FUNCTION_BLOCK RunCableHolder EXTENDS RunUnitSlave
VAR
	//devices
	holderFixedEnd : POINTER TO RunCylinder;
	holderMovingEnd : POINTER TO RunCylinder;
	shifterShort : POINTER TO RunCylinder;
	shifterLong : POINTER TO RunCylinder;
	//axis (share
	axis : POINTER TO RunAxis;
	ptDrag : POINTER TO ParameterSet;
	ptRelease : pointer to ParameterSet;
END_VAR

SUPER^();

CASE outputState OF
	//---------------Initialize
	eSpecialStates.INITIAL_BEGIN:
		transitionByte.0 :=  holderFixedEnd^.Execute(eCylinderCommands.COMMAND_A);
		transitionByte.1 :=  holderMovingEnd^.Execute(eCylinderCommands.COMMAND_A);
		transitionByte.2 :=  shifterShort^.Execute(eCylinderCommands.COMMAND_A);
		transitionByte.3 :=  shifterLong^.Execute(eCylinderCommands.COMMAND_A);
		IF transitionByte = 16#F THEN
			NextState := eSpecialStates.INITIAL_END;
		END_IF
	//---------------Working
	eSpecialStates.SLAVE_ENTER_PROCEDURE:
		IF SlotBase^.Valid THEN
			bSerialTransition := TRUE;
		ELSE
			NextState := eSpecialStates.SLAVE_WORK_DONE;	
		END_IF
		//TODO , check ok/ng?
	16#201:
		bSerialTransition := shifterLong^.Execute(eCylinderCommands.COMMAND_B);
	16#202:
		//hold
		transitionByte.0 :=  holderFixedEnd^.Execute(eCylinderCommands.COMMAND_B);
		transitionByte.1 :=  holderMovingEnd^.Execute(eCylinderCommands.COMMAND_B);
		bSerialTransition := (transitionByte = 16#3);
	16#203:
		bSerialTransition := axis^.ExecuteParameter(ptDrag);//inform transporter moving work2
	16#204:
		//strech
		IF shifterShort^.Execute(eCylinderCommands.COMMAND_B) THEN
			slaveWorkingSignal[1] := TRUE; //inform to labeler handler to work
			NextState := 16#210;
		END_IF
	//-------------Releasing
	16#210:
		//wait until
		bSerialTransition := NOT slaveWorkingSignal[1];
	16#211:
		transitionByte.0 := holderFixedEnd^.Execute(eCylinderCommands.COMMAND_A); //release
		transitionByte.1 := holderMovingEnd^.Execute(eCylinderCommands.COMMAND_A);
		IF transitionByte = 16#3 THEN
			bSerialTransition := TRUE;
		END_IF
	16#212:
		bSerialTransition := axis^.ExecuteParameter(ptRelease);//inform transporter moving release
	16#213:
		//release
		bSerialTransition := shifterLong^.Execute(eCylinderCommands.COMMAND_A);
	16#214:
		//release
		bSerialTransition := holderMovingEnd^.Execute(eCylinderCommands.COMMAND_A);
	16#215:
		IF shifterShort^.Execute(eCylinderCommands.COMMAND_A) THEN
			NextState := eSpecialStates.SLAVE_WORK_DONE; //rewind
		END_IF
END_CASE

METHOD FB_init : BOOL
VAR_INPUT
	bInitRetains : BOOL; // if TRUE, the retain variables are initialized (warm start / cold start)
	bInCopyCode : BOOL;  // if TRUE, the instance afterwards gets moved into the copy code (online change)
	
	argParent : POINTER TO RunUnitGeneric;
	argSlotBase : POINTER TO RunMaterial;
	argSlotLast : POINTER TO RunMaterial;
	
	argWorkingSignal : POINTER TO BOOL;
	
	//devices
	argHolderFixedEnd : POINTER TO RunCylinder;
	argHolderMovingEnd : POINTER TO RunCylinder;
	argShifterShort : POINTER TO RunCylinder;
	argShifterLong : POINTER TO RunCylinder;
	
	//
	argAxis : POINTER TO RunAxis;
END_VAR
VAR CONSTANT
	indexDrag : INT :=8;
	indexRelease : int :=9;
END_VAR
//initialize 
Parent := argParent;
SlotBase := argSlotBase;
SlotLast := argSlotLast;
//
IF bInitRetains THEN
	NextState := eSpecialStates.INITIAL_BEGIN;
END_IF

workingSignal := argWorkingSignal; //link

//device link
holderFixedEnd := argHolderFixedEnd;
holderMovingEnd := argHolderMovingEnd;
shifterShort := argShifterShort;
shifterLong := argShifterLong;

//
axis := argAxis;
ptDrag := ADR(axis^.ptpCommands[indexDrag]);
ptRelease := ADR(axis^.ptpCommands[indexRelease]);
END_METHOD

END_FUNCTION_BLOCK

(* stored: Version 1.1.0.1, ProductVersion 3.1.4022.10
   POU RunCableHolder: Id {f529174f-1b1c-4098-af22-9f3935583d60}, SpecialFunc None
   Method FB_init: Id {5c2d8834-883b-4bdd-9d6d-567f106a2a04} *)
